// TIA Portal V17 export
// export: Created 2022-07-28T18:02:49.0040858Z, ExportSetting None, DisplayName Totally Integrated Automation Portal, DisplayVersion V17, DisplayName TIA Portal Openness, DisplayVersion V17, DisplayName TIA Portal Teamcenter Gateway, DisplayVersion V17, DisplayName TIA Portal Version Control Interface, DisplayVersion V17, DisplayName TIA Portal Test Suite Advanced, DisplayVersion V17, DisplayName SINAMICS Startdrive Advanced, DisplayVersion V17, DisplayName SINAMICS DCC, DisplayVersion V17, DisplayName SINAMICS Startdrive G130, G150, S120, S150, SINAMICS MV, S210, DisplayVersion V17, DisplayName SINAMICS Startdrive G110M, G120, G120C, G120D, G120P, G115D, DisplayVersion V17, DisplayName STEP 7 Professional, DisplayVersion V17, DisplayName SIMATIC Energy Suite, DisplayVersion V17, DisplayName STEP 7 CFC, DisplayVersion V17, DisplayName STEP 7 Safety, DisplayVersion V17, DisplayName WinCC Advanced / Unified PC, DisplayVersion V17, DisplayName SIMATIC Visualization Architect, DisplayVersion V17
FUNCTION_BLOCK "Lib_FB_PID_Cascad"   // FB151, SCL
{ S7_Optimized_Access := 'TRUE' }
// stored: AutoNumber false, MemoryReserve 100, SetENOAutomatically false
   VAR_INPUT
      I_Initialization { ExternalAccessible := 'False'; ExternalVisible := 'False'; ExternalWritable := 'False'} : Bool := FALSE;   // 1 = Restart PLC is active (First scan)
      IR_CycleTime { ExternalAccessible := 'False'; ExternalVisible := 'False'; ExternalWritable := 'False'} : Real := 0.0;   // Time of last PLC cycle, sec
      II_Obj_ID { ExternalAccessible := 'False'; ExternalVisible := 'False'; ExternalWritable := 'False'} : Int := -1;   // Tech ID of object
      I_CmdGeneralReset { ExternalAccessible := 'False'; ExternalVisible := 'False'; ExternalWritable := 'False'} : Bool;   // 0 ⮥ 1 = Input general reset ERROR/Interlocks
      I_One_1s { ExternalAccessible := 'False'; ExternalVisible := 'False'; ExternalWritable := 'False'} : Bool;   // 1 = One cycle per one seccond pulse
      I_EstopHMI { ExternalAccessible := 'False'; ExternalVisible := 'False'; ExternalWritable := 'False'} : Bool := TRUE;   // 0 = HMI/WinCC Emergency stop active
      IR_SP_Auto { ExternalAccessible := 'False'; ExternalVisible := 'False'; ExternalWritable := 'False'} : Real;   // SP for auto mode from input in physics units
      IR_MinOut { ExternalAccessible := 'False'; ExternalVisible := 'False'; ExternalWritable := 'False'} : Real := 15.0;   // Minimum output of PID, PU
      IR_MaxOut { ExternalAccessible := 'False'; ExternalVisible := 'False'; ExternalWritable := 'False'} : Real := 100.0;   // Maximum output of PID, PU
      IB_InterlocksOpen_8 { ExternalAccessible := 'False'; ExternalVisible := 'False'; ExternalWritable := 'False'} : Byte;   // <>0 = Interlock active - One or more from 8 Interlocks active // 1bit <--> 1 Interlock
      IB_InterlocksClose_8 { ExternalAccessible := 'False'; ExternalVisible := 'False'; ExternalWritable := 'False'} : Byte;   // <>0 = Interlock active - One or more from 8 Interlocks active // 1bit <--> 1 Interlock
      IW_ExternalError_16 { ExternalAccessible := 'False'; ExternalVisible := 'False'; ExternalWritable := 'False'} : Word;   // <>0 = External error active - One or more from 16 error active // 1bit <--> 1 error
      I_ExternalWarning { ExternalAccessible := 'False'; ExternalVisible := 'False'; ExternalWritable := 'False'} : Bool;   // 1 = External Warning
      IR_CyclePID { ExternalAccessible := 'False'; ExternalVisible := 'False'; ExternalWritable := 'False'} : Real;   // Cycle tyme of PID, sec
      II_ID_Sensor { ExternalAccessible := 'False'; ExternalVisible := 'False'; ExternalWritable := 'False'} : Int := -1;   // ID of sensor for PID
      IA_ID_Inv { ExternalAccessible := 'False'; ExternalVisible := 'False'; ExternalWritable := 'False'} : Array[0..5] of Int;   // IDs of inverters for PID
      II_Num_Inv { ExternalAccessible := 'False'; ExternalVisible := 'False'; ExternalWritable := 'False'} : Int := 3;   // Numbers of inverters
   END_VAR
   VAR_OUTPUT
      QR_Out_PID { ExternalAccessible := 'False'; ExternalVisible := 'False'; ExternalWritable := 'False'} : Real;   // Output of PID in physics unit (0-100%)
      QI_Out_PID { ExternalAccessible := 'False'; ExternalVisible := 'False'; ExternalWritable := 'False'} : Int;   // Output of PID in analog output units (0-27648)
      Q_CmdPWM { ExternalAccessible := 'False'; ExternalVisible := 'False'; ExternalWritable := 'False'} : Bool;   // PWM signal for descrete output mechanism
      Q_Reset { ExternalAccessible := 'False'; ExternalVisible := 'False'; ExternalWritable := 'False'} : Bool;   // 1 = Reset faults
      Q_Error { ExternalAccessible := 'False'; ExternalVisible := 'False'; ExternalWritable := 'False'} : Bool;   // This output indicates whether theres an error/fault condition in the motor
      Q_Auto { ExternalAccessible := 'False'; ExternalVisible := 'False'; ExternalWritable := 'False'} : Bool;   // 1= Automatic operating mode active
      Q_DataErr { ExternalAccessible := 'False'; ExternalVisible := 'False'; ExternalWritable := 'False'} : Bool;   // 1 = Transfer data error occured (ObjDB -> temp, ect)
   END_VAR
   VAR_IN_OUT
      IQ_PLC_CycleInfo : Variant;   // Ref to data about PLC cycle
   END_VAR
   VAR
      s_ErrForSwitchToOff { ExternalAccessible := 'False'; ExternalVisible := 'False'; ExternalWritable := 'False'} : Bool;   // 1 = Err occured for switch to manual mode
   END_VAR
   VAR RETAIN
      si_OldPriority_P1 { ExternalAccessible := 'False'; ExternalVisible := 'False'; ExternalWritable := 'False'} : Int := 1;
      si_OldPriority_P2 { ExternalAccessible := 'False'; ExternalVisible := 'False'; ExternalWritable := 'False'} : Int := 2;
      si_OldPriority_P3 { ExternalAccessible := 'False'; ExternalVisible := 'False'; ExternalWritable := 'False'} : Int := 3;
   END_VAR
   VAR
      si_CurrentPIDPoint { ExternalAccessible := 'False'; ExternalVisible := 'False'; ExternalWritable := 'False'} : Int;
      si_PrevPIDPoint { ExternalAccessible := 'False'; ExternalVisible := 'False'; ExternalWritable := 'False'} : Int;
      s_EdgeAuto { ExternalAccessible := 'False'; ExternalVisible := 'False'; ExternalWritable := 'False'} : "Lib_FB_Edge";
      s_EdgeMan { ExternalAccessible := 'False'; ExternalVisible := 'False'; ExternalWritable := 'False'} : "Lib_FB_Edge";
      s_EdgeOff { ExternalAccessible := 'False'; ExternalVisible := 'False'; ExternalWritable := 'False'} : "Lib_FB_Edge";
      s_EdgeSim { ExternalAccessible := 'False'; ExternalVisible := 'False'; ExternalWritable := 'False'} : "Lib_FB_Edge";
      s_EdgeError { ExternalAccessible := 'False'; ExternalVisible := 'False'; ExternalWritable := 'False'} : "Lib_FB_Edge";
      s_EdgeWarning { ExternalAccessible := 'False'; ExternalVisible := 'False'; ExternalWritable := 'False'} : "Lib_FB_Edge";
      s_EdgeUp { ExternalAccessible := 'False'; ExternalVisible := 'False'; ExternalWritable := 'False'} : "Lib_FB_Edge";
      s_EdgeDwn { ExternalAccessible := 'False'; ExternalVisible := 'False'; ExternalWritable := 'False'} : "Lib_FB_Edge";
   END_VAR
   VAR RETAIN
      s_Simulation { ExternalAccessible := 'False'; ExternalVisible := 'False'; ExternalWritable := 'False'} : Struct   // Data for simulation process
         Obj_DATA_BACKUP : Struct   // MOTOR NORMAL MODE DATA BACKUP FOR SIMULATION MODE
            Config : "_PID_Cascad_Config";
            Counters : "_PID_Cascad_Counters";
            sud_MotoHours_Electro : "_MotoHours_One";
            sud_MotoHours_Mech : "_MotoHours_One";
         END_STRUCT;
      END_STRUCT;
      s_Obj_Retain_BUp { ExternalAccessible := 'False'; ExternalVisible := 'False'; ExternalWritable := 'False'} : Struct
         Config : "_PID_Cascad_Config";
         Counters : "_PID_Cascad_Counters";
         Mode : "UDT_Mode";
      END_STRUCT;
   END_VAR
   VAR
      s_TP_ResetOut { ExternalAccessible := 'False'; ExternalVisible := 'False'; ExternalWritable := 'False'} : "Lib_FB_Timer_TP_Simple";
      s_TON_TimeUP { ExternalAccessible := 'False'; ExternalVisible := 'False'; ExternalWritable := 'False'} : "Lib_FB_Timer_ON_Simple";
      s_TON_TimeDwn { ExternalAccessible := 'False'; ExternalVisible := 'False'; ExternalWritable := 'False'} : "Lib_FB_Timer_ON_Simple";
      s_TON_Stabilization { ExternalAccessible := 'False'; ExternalVisible := 'False'; ExternalWritable := 'False'} : "Lib_FB_Timer_ON_Simple";
   END_VAR
   VAR_TEMP
      t_DataErr : Bool;   // 1 = Transfer data error occured (ObjDB -> temp, ect)
      t_ReleaseStart : Bool;   // 1 = Release for start in any mode
      t_SomePumpIsRunning : Bool;
      t_ResetLogic : Bool;   // 1 = Reset all signals for logic
      ti_CMDLogic : Int;   // Command word for logic
      ti_Cnt : Int;   // Counter for internal use
      ti_NumObjDB : UInt;   // Number of DB for storage object data
      t_MaxObjects : UInt;   // Max number of objects in plant
      tr_PID_Out : Real;   // SP in auto mode for logic
      tr_InvertCoef : Real;
      t_ObjAny_PIDCon : DB_ANY;
      t_ObjVar_PIDCon : Variant;
      t_ObjAny_HMI : DB_ANY;   // Ref to object data
      t_ObjVar_HMI : Variant;   // Ref to object data
      t_ObjAny_PLC : DB_ANY;   // Ref to object data
      t_ObjVar_PLC : Variant;   // Ref to object data
      t_SensorObjAny_HMI : DB_ANY;   // Ref to object data
      t_SensorObjVar_HMI : Variant;   // Ref to object data
      t_Pump1_ObjAny_HMI : DB_ANY;   // Ref to object data
      t_Pump1_ObjVar_HMI : Variant;   // Ref to object data
      t_Pump2_ObjAny_HMI : DB_ANY;   // Ref to object data
      t_Pump2_ObjVar_HMI : Variant;   // Ref to object data
      t_Pump3_ObjAny_HMI : DB_ANY;   // Ref to object data
      t_Pump3_ObjVar_HMI : Variant;   // Ref to object data
      t_PB_HMI : Struct   // Buttons from HMI
         ResetError : Bool;   // + set-->CMD_ALMACK_tag -Reset errors pushbutton
         AllInAuto : Bool;   // 1 = All pumps switch to auto
         spare2 : Bool;
         spare3 : Bool;
         spare4 : Bool;
         spare5 : Bool;
         spare6 : Bool;
         spare7 : Bool;
         spare8 : Bool;
         spare9 : Bool;
         spare10 : Bool;
         spare11 : Bool;
         spare12 : Bool;
         spare13 : Bool;
         spare14 : Bool;
         spare15 : Bool;
         spare16 : Bool;
         spare17 : Bool;
         spare18 : Bool;
         spare19 : Bool;
         spare20 : Bool;
         spare21 : Bool;
         spare22 : Bool;
         spare23 : Bool;
         spare24 : Bool;
         spare25 : Bool;
         spare26 : Bool;
         spare27 : Bool;
         spare28 : Bool;
         spare29 : Bool;
         spare30 : Bool;
         spare31 : Bool;
      END_STRUCT;
      t_Obj_HMI : "Lib_UDT_PID_Cascad_HMI";   // Object data
      t_Obj_PLC : "Lib_UDT_PID_Cascad_PLC";   // Object data
      t_Obj_PIDCon : "Lib_UDT_PID_Core";
      t_SensorObj_HMI : "lib_udt_ASensor_HMI";   // Object data
      t_Pump1_Obj_HMI : "Lib_UDT_Pump_Inv352_Base_HMI";   // Object data
      t_Pump2_Obj_HMI : "Lib_UDT_Pump_Inv352_Base_HMI";   // Object data
      t_Pump3_Obj_HMI : "Lib_UDT_Pump_Inv352_Base_HMI";   // Object data
      t_PLC_CycleInfo : "Lib_PLC_CycleInfo";   // Data about PLC cycle
      t_AutoControl : "Lib_UDT_AutoControl";   // Data for auto control module for current element
      t_AutoControl_Pumps : "_PID_Cascad_AutoCtrlPumpsAll";   // Data for auto control module for current element
      t_AutoControl_Pumps_Sorted : "_PID_Cascad_AutoCtrlPumpsAll";   // Data for auto control module for current element
      t_InternalData : "Lib_UDT_Int";   // Internal data
      t_Buffer : Array[0..100] of Byte;   // Buffer for use serialize
      tui_DB_ShiftHMI : UInt;   // Object DB number shift
      tui_DB_ShiftPLC : UInt;   // Object DB number shift
      tui_DB_ShiftPID : UInt;
   END_VAR
   // IA_ID_Inv[0..5] := -1;
BEGIN
   REGION Initialization/read data from out DB
       //Set internal data
       "Lib_FC_GenMoto_InitInternal"(#t_InternalData);

       //Reinit gen data
       #t_DataErr := false;
       #t_Obj_HMI.Config.w_enableExternalErrors_16 := w#16#FFFF;
       #t_Obj_HMI.Config.b_bypassInterlocksForward_8 := b#16#ff;
       #t_Obj_HMI.Config.b_bypassInterlocksReverse_8 := b#16#ff;
       #t_MaxObjects := "D_General_ProgramDATA".ui_MaxObjects;
       #tui_DB_ShiftHMI := "D_General_ProgramDATA".ui_Shift_DB_HMI;
       #tui_DB_ShiftPLC := "D_General_ProgramDATA".ui_Shift_DB_PLC;
       #tui_DB_ShiftPID := "D_General_ProgramDATA".ui_Shift_DB_PID;
       #t_AutoControl := "DB_AutoControl_arr".AutoControl_arr[#t_MaxObjects];
       #t_AutoControl_Pumps.Arr[0].AutoControl_P := "DB_AutoControl_arr".AutoControl_arr[#t_MaxObjects];
       #t_AutoControl_Pumps.Arr[1].AutoControl_P := "DB_AutoControl_arr".AutoControl_arr[#t_MaxObjects];
       #t_AutoControl_Pumps.Arr[2].AutoControl_P := "DB_AutoControl_arr".AutoControl_arr[#t_MaxObjects];

       //Read data PLC
       VariantGet(SRC := #IQ_PLC_CycleInfo,
                  DST => #t_PLC_CycleInfo);

       //Read Object data
       //Reinit temp values
       #t_Obj_HMI := "D_ZeroTypes".PID_Cascad_HMI;
       #t_Obj_PLC := "D_ZeroTypes".PID_Cascad_PLC;
       #t_SensorObj_HMI := "D_ZeroTypes".ASensor_HMI;
       #t_Pump1_Obj_HMI := "D_ZeroTypes".Pump_Inv352_Base_HMI;
       #t_Pump2_Obj_HMI := "D_ZeroTypes".Pump_Inv352_Base_HMI;
       #t_Pump3_Obj_HMI := "D_ZeroTypes".Pump_Inv352_Base_HMI;
       #t_Obj_PIDCon := "D_ZeroTypes".PID_Core;

       //Read object data
       IF #II_Obj_ID >= 0
       THEN
           //Read HMI data
           #ti_NumObjDB := INT_TO_UINT(#II_Obj_ID) + #tui_DB_ShiftHMI;
           #t_ObjAny_HMI := UINT_TO_DB_ANY(#ti_NumObjDB);
           #t_ObjVar_HMI := DB_ANY_TO_VARIANT(in := #t_ObjAny_HMI, err => #t_InternalData.i_Tmp);

           //If DB exist and convertion without error
           IF #t_InternalData.i_Tmp = 0
           THEN
               VariantGet(SRC := #t_ObjVar_HMI,
                          DST => #t_Obj_HMI);
           ELSE
               #t_DataErr := true;
           END_IF;

           //Read PLC data
           #ti_NumObjDB := INT_TO_UINT(#II_Obj_ID) + #tui_DB_ShiftPLC;
           #t_ObjAny_PLC := UINT_TO_DB_ANY(#ti_NumObjDB);
           #t_ObjVar_PLC := DB_ANY_TO_VARIANT(in := #t_ObjAny_PLC, err => #t_InternalData.i_Tmp);

           //If DB exist and convertion without error
           IF #t_InternalData.i_Tmp = 0
           THEN
               VariantGet(SRC := #t_ObjVar_PLC,
                          DST => #t_Obj_PLC);
           ELSE
               #t_DataErr := true;
           END_IF;

           //Read PID data
           #ti_NumObjDB := INT_TO_UINT(#II_Obj_ID) + #tui_DB_ShiftPID;
           #t_ObjAny_PIDCon := UINT_TO_DB_ANY(#ti_NumObjDB);
           #t_ObjVar_PIDCon := DB_ANY_TO_VARIANT(in := #t_ObjAny_PIDCon, err => #t_InternalData.i_Tmp);

           //If DB exist and convertion without error
           IF #t_InternalData.i_Tmp = 0
           THEN
               VariantGet(SRC := #t_ObjVar_PIDCon,
                          DST => #t_Obj_PIDCon);
           ELSE
               #t_DataErr := true;
           END_IF;
       ELSE
           #t_DataErr := true;
       END_IF;

       //Read sensor data
       IF #II_ID_Sensor >= 0
           AND NOT #t_DataErr
       THEN
           //Read HMI data
           #ti_NumObjDB := INT_TO_UINT(#II_ID_Sensor) + 50000;
           #t_SensorObjAny_HMI := UINT_TO_DB_ANY(#ti_NumObjDB);
           #t_SensorObjVar_HMI := DB_ANY_TO_VARIANT(in := #t_SensorObjAny_HMI, err => #t_InternalData.i_Tmp);

           //If DB exist and convertion without error
           IF #t_InternalData.i_Tmp = 0
           THEN
               VariantGet(SRC := #t_SensorObjVar_HMI,
                          DST => #t_SensorObj_HMI);
           ELSE
               #t_DataErr := true;
           END_IF;
       ELSE
           #t_DataErr := true;
       END_IF;

       //Read pumps data
       IF #IA_ID_Inv[0] >= 0
           AND NOT #t_DataErr
       THEN
           REGION Pump 1
               //Read HMI data
               #ti_NumObjDB := INT_TO_UINT(#IA_ID_Inv[0]) + #tui_DB_ShiftHMI;
               #t_Pump1_ObjAny_HMI := UINT_TO_DB_ANY(#ti_NumObjDB);
               #t_Pump1_ObjVar_HMI := DB_ANY_TO_VARIANT(in := #t_Pump1_ObjAny_HMI, err => #t_InternalData.i_Tmp);

               //If DB exist and convertion without error
               IF #t_InternalData.i_Tmp = 0
               THEN
                   VariantGet(SRC := #t_Pump1_ObjVar_HMI,
                              DST => #t_Pump1_Obj_HMI);
               ELSE
                   #t_DataErr := true;
               END_IF;

               #t_AutoControl_Pumps.Arr[0].AutoControl_P := "DB_AutoControl_arr".AutoControl_arr[#IA_ID_Inv[0]];
               #t_AutoControl_Pumps.Arr[0].i_IndexInArr := 0;
           END_REGION

       ELSE
           #t_DataErr := true;
       END_IF;

       IF #IA_ID_Inv[1] >= 0
           AND NOT #t_DataErr
       THEN
           REGION Pump 2
               //Read HMI data
               #ti_NumObjDB := INT_TO_UINT(#IA_ID_Inv[1]) + #tui_DB_ShiftHMI;
               #t_Pump2_ObjAny_HMI := UINT_TO_DB_ANY(#ti_NumObjDB);
               #t_Pump2_ObjVar_HMI := DB_ANY_TO_VARIANT(in := #t_Pump2_ObjAny_HMI, err => #t_InternalData.i_Tmp);

               //If DB exist and convertion without error
               IF #t_InternalData.i_Tmp = 0
               THEN
                   VariantGet(SRC := #t_Pump2_ObjVar_HMI,
      DST => #t_Pump2_Obj_HMI);
               ELSE
                   #t_DataErr := true;
               END_IF;

               #t_AutoControl_Pumps.Arr[1].AutoControl_P := "DB_AutoControl_arr".AutoControl_arr[#IA_ID_Inv[1]];
               #t_AutoControl_Pumps.Arr[1].i_IndexInArr := 1;
           END_REGION

       ELSE
           #t_DataErr := true;
       END_IF;

       IF #IA_ID_Inv[2] >= 0
           AND NOT #t_DataErr
       THEN
           REGION Pump 3
               //Read HMI data
               #ti_NumObjDB := INT_TO_UINT(#IA_ID_Inv[2]) + #tui_DB_ShiftHMI;
               #t_Pump3_ObjAny_HMI := UINT_TO_DB_ANY(#ti_NumObjDB);
               #t_Pump3_ObjVar_HMI := DB_ANY_TO_VARIANT(in := #t_Pump3_ObjAny_HMI, err => #t_InternalData.i_Tmp);

               //If DB exist and convertion without error
               IF #t_InternalData.i_Tmp = 0
               THEN
                   VariantGet(SRC := #t_Pump3_ObjVar_HMI,
      DST => #t_Pump3_Obj_HMI);
               ELSE
                   #t_DataErr := true;
               END_IF;

               #t_AutoControl_Pumps.Arr[2].AutoControl_P := "DB_AutoControl_arr".AutoControl_arr[#IA_ID_Inv[2]];
               #t_AutoControl_Pumps.Arr[2].i_IndexInArr := 2;
           END_REGION
       ELSE
           #t_DataErr := true;
       END_IF;

       //Read general info data
       CASE #II_Obj_ID OF
           0..999:  // ID of element in range
               #t_AutoControl := "DB_AutoControl_arr".AutoControl_arr[#II_Obj_ID];
           ELSE
               ;
       END_CASE;

       //Read retain data if initialization is active
       IF #I_Initialization
       THEN
           #t_Obj_HMI.Config := #s_Obj_Retain_BUp.Config;
           #t_Obj_HMI.Counters := #s_Obj_Retain_BUp.Counters;
           #t_Obj_PLC.Mode := #s_Obj_Retain_BUp.Mode;
       END_IF;
   END_REGION
   //---------------------------------------------------------------
   //---------------------------------------------------------------
   REGION Check ranges
       //Invert coef
       IF #t_Obj_HMI.Config.b.DirectMode
       THEN
           #tr_InvertCoef := 1.0;
       ELSE
           #tr_InvertCoef := -1.0;
       END_IF;

       IF #t_Obj_HMI.Config.r_FTC_Value > #IR_MaxOut
       THEN
           #t_Obj_HMI.Config.r_FTC_Value := #IR_MaxOut;
       END_IF;

       IF #t_Obj_HMI.Config.r_FTC_Value < #IR_MinOut
       THEN
           #t_Obj_HMI.Config.r_FTC_Value := #IR_MinOut;
       END_IF;

       IF #t_Obj_HMI.Config.r_SP_Auto_Value > #t_SensorObj_HMI.Config.r_MaxVal
       THEN
           #t_Obj_HMI.Config.r_SP_Auto_Value := #t_SensorObj_HMI.Config.r_MaxVal;
       END_IF;

       IF #t_Obj_HMI.Config.r_SP_Auto_Value < #t_SensorObj_HMI.Config.r_MinVal
       THEN
           #t_Obj_HMI.Config.r_SP_Auto_Value := #t_SensorObj_HMI.Config.r_MinVal;
       END_IF;
   END_REGION
   //---------------------------------------------------------------
   //---------------------------------------------------------------
   REGION Define CMD for block logic 
       //Reinit logic CMD
       #ti_CMDLogic := 0;

       "Lib_FC_GenMoto_ChoiceCMD"(I_Mode := #t_Obj_PLC.Mode,
                                  QI_CMD_Logic => #ti_CMDLogic,
                                  IQI_CMD_Global := #t_PLC_CycleInfo.CMD_GLOBAL,
                                  IQI_CMD_Auto := #t_AutoControl.Global_CMD,
                                  IQI_CMD_HMI := #t_Obj_HMI.i_CMD);

   END_REGION
   //---------------------------------------------------------------
   //---------------------------------------------------------------
   REGION Switch modes  
       "Lib_FC_GenMoto_SwitchMode"(I_ManLocalModeActive := false,
                                   IQI_CMD_Logic := #ti_CMDLogic,
                                   IQ_Mode := #t_Obj_PLC.Mode,
                                   IQ_ObjDataConfig := #t_Obj_HMI.Config,
                                   IQ_BUpDataConfig := #s_Simulation.Obj_DATA_BACKUP.Config,
                                   IQ_ObjDataCounters := #t_Obj_HMI.Counters,
                                   IQ_BUpDataCounters := #s_Simulation.Obj_DATA_BACKUP.Counters);
                                END_REGION
   //---------------------------------------------------------------
   //---------------------------------------------------------------
   REGION Forcely switch modes by mode of PID  
      (* 
       IF (NOT (#t_Obj_PIDCon.i_State = 4)
           AND NOT (#t_Obj_PIDCon.i_State = 3))
           OR #s_ErrForSwitchToOff
       THEN
           #ti_CMDLogic := 1;
       END_IF;

       "Lib_FC_GenMoto_SwitchMode"(I_ManLocalModeActive := false,
                                   IQI_CMD_Logic := #ti_CMDLogic,
                                   IQ_Mode := #t_Obj_PLC.Mode,
                                   IQ_ObjDataConfig := #t_Obj_HMI.Config,
                                   IQ_BUpDataConfig := #s_Simulation.Obj_DATA_BACKUP.Config,
                                   IQ_ObjDataCounters := #t_Obj_HMI.Counters,
                                   IQ_BUpDataCounters := #s_Simulation.Obj_DATA_BACKUP.Counters); *)
   END_REGION
   //---------------------------------------------------------------
   //---------------------------------------------------------------
   REGION Convert commands to bit
       //Reinit all bits
       SCATTER(IN := #t_InternalData.d_Alw0,
               OUT => #t_PB_HMI);

       //Read commands and set apropriate bits
       CASE #ti_CMDLogic OF
           22:  //Direct mode
               #t_Obj_HMI.Config.b.DirectMode := true;
           23:  //Invert mode
               #t_Obj_HMI.Config.b.DirectMode := false;
           24:  //Invert mode
               #t_Obj_HMI.Config.b.Enabled_P1 := true;
           25:  //Invert mode
               #t_Obj_HMI.Config.b.Enabled_P2 := true;
           26:  //Invert mode
               #t_Obj_HMI.Config.b.Enabled_P3 := true;
           27:  //Invert mode
               #t_Obj_HMI.Config.b.Enabled_P1 := false;
           28:  //Invert mode
               #t_Obj_HMI.Config.b.Enabled_P2 := false;
           29:  //Invert mode
               #t_Obj_HMI.Config.b.Enabled_P3 := false;
           31..32: // Reset errors
               #t_PB_HMI.ResetError := true;
           30:// Switch all pumps to auto
               #t_PB_HMI.AllInAuto := true;

           ELSE
               ;
       END_CASE;

       //General bits for logic
       //General reset
       #t_ResetLogic := #t_PB_HMI.ResetError
       OR #I_CmdGeneralReset;

       //Reset for out of block
       #s_TP_ResetOut(IR_CycleTime := #IR_CycleTime,
                      IB_StartTimerInput := #t_ResetLogic,
                      IR_SpTime := 1.5);

                   END_REGION
   //---------------------------------------------------------------
   //---------------------------------------------------------------
   REGION Switch mode on PID
       //Catch change mode
       #s_EdgeAuto(IB_Input := #t_Obj_PLC.Mode.Auto);
       #s_EdgeMan(IB_Input := #t_Obj_PLC.Mode.ManualRemote);
       #s_EdgeOff(IB_Input := #s_ErrForSwitchToOff);

       IF #s_EdgeAuto.QB_EdgePos
           OR #s_EdgeMan.QB_EdgePos
           OR #s_EdgeOff.QB_EdgePos
       THEN
           #t_Obj_PIDCon.ModeActivate := true;
       END_IF;
       //Set value for auto mode
       IF (#s_EdgeAuto.QB_EdgePos
           AND #t_Obj_PIDCon.ModeActivate
           AND NOT (#t_Obj_PIDCon.i_State = 3))
       THEN
           #t_Obj_PIDCon.i_Mode := 3;
       END_IF;

       //Set value for manual mode
       IF (#s_EdgeMan.QB_EdgePos
           AND #t_Obj_PIDCon.ModeActivate
           AND NOT (#t_Obj_PIDCon.i_State = 4))
       THEN
           #t_Obj_PIDCon.i_Mode := 4;
       END_IF;

       //Set value for off mode
       IF (#s_EdgeOff.QB_EdgePos
           AND #t_Obj_PIDCon.ModeActivate
           AND NOT (#t_Obj_PIDCon.i_State = 0))
       THEN
           #t_Obj_PIDCon.i_Mode := 0;
       END_IF;
   END_REGION
   //---------------------------------------------------------------
   //---------------------------------------------------------------
   REGION Write data to PID and call him
       #t_Obj_PIDCon.r_Setpoint := #t_Obj_HMI.Config.r_SP_Auto_Value;
       #t_Obj_PIDCon.r_ManualValue := #t_Obj_HMI.Config.r_SP_Man_Value;
       #t_Obj_PIDCon.r_Input := #t_SensorObj_HMI.Config.r_DisplayData;
       IF #t_ResetLogic
       THEN
           #t_Obj_PIDCon.ErrorAck := true;
       END_IF;
       IF #I_Initialization
       THEN
           #t_Obj_PIDCon.Reset := true;
       END_IF;
       #t_Obj_PIDCon.r_OutputUpperLimit := #IR_MaxOut;
       #t_Obj_PIDCon.r_OutputLowerLimit := #IR_MinOut;
       #t_Obj_PIDCon.r_CycleTime_Value := #IR_CyclePID;
       #t_Obj_PIDCon.r_Gain := #tr_InvertCoef * #t_Obj_HMI.Config.r_spP_part;
       #t_Obj_PIDCon.r_Ti := #t_Obj_HMI.Config.r_spI_part;
       #t_Obj_PIDCon.r_Td := #t_Obj_HMI.Config.r_spD_part;
       #t_Obj_PIDCon.InvertControl := false; //NOT #t_Obj_HMI.Config.b.DirectMode;
       #t_Obj_PIDCon.r_SPUpperLimit := #t_SensorObj_HMI.Config.r_MaxVal;
       #t_Obj_PIDCon.r_SPLowerLimit := #t_SensorObj_HMI.Config.r_MinVal;
       #t_Obj_PIDCon.r_PVUpperLimit := #t_SensorObj_HMI.Config.r_MaxVal;
       #t_Obj_PIDCon.r_PVLowerLimit := #t_SensorObj_HMI.Config.r_MinVal;
       #t_Obj_PIDCon.r_Cycle_PID := 1.0;

       //Write mode by mode on PID
       #t_Obj_PLC.Mode.Auto := #t_Obj_PIDCon.i_State = 3;
       #t_Obj_PLC.Mode.ManualRemote := #t_Obj_PIDCon.i_State = 4;
       #t_Obj_PLC.Mode.Disable := #t_Obj_PIDCon.i_State = 0;

       REGION Store out of PID in temp var dependent of state
           IF #t_Obj_PIDCon.i_State = 3
               OR #t_Obj_PIDCon.i_State = 4
           THEN
               #tr_PID_Out := #t_Obj_PIDCon.r_Output;
           ELSE
               IF #t_Obj_PLC.State.FTCActive
               THEN
                   #tr_PID_Out := #t_Obj_HMI.Config.r_FTC_Value;
               ELSIF #t_Obj_PLC.State.FTOActive
               THEN
                   #tr_PID_Out := #t_Obj_HMI.Config.r_FTO_Value;
               ELSE
                   #tr_PID_Out := #IR_MinOut;
               END_IF;
           END_IF;
       END_REGION

   END_REGION
   //---------------------------------------------------------------
   //---------------------------------------------------------------
   REGION Control of pumps

       REGION Define number OF enabled pumps
           #t_Obj_HMI.Config.r_QuanEnabled := 0;

           IF #t_Obj_HMI.Config.b.Enabled_P1
           THEN
               #t_Obj_HMI.Config.r_QuanEnabled := #t_Obj_HMI.Config.r_QuanEnabled + 1;
           END_IF;
           IF #t_Obj_HMI.Config.b.Enabled_P2
           THEN
               #t_Obj_HMI.Config.r_QuanEnabled := #t_Obj_HMI.Config.r_QuanEnabled + 1;
           END_IF;
           IF #t_Obj_HMI.Config.b.Enabled_P3
           THEN
               #t_Obj_HMI.Config.r_QuanEnabled := #t_Obj_HMI.Config.r_QuanEnabled + 1;
           END_IF;

       END_REGION

       REGION Define priority of pumps
           IF #t_Obj_HMI.Config.b.Enabled_P1
           THEN
               IF #t_Obj_HMI.Config.i_Priority_P1 > #t_Obj_HMI.Config.r_QuanEnabled
               THEN
                   #t_Obj_HMI.Config.i_Priority_P1 := #t_Obj_HMI.Config.r_QuanEnabled;
                   #si_OldPriority_P1 := #t_Obj_HMI.Config.r_QuanEnabled;
               END_IF;
           ELSE
               #t_Obj_HMI.Config.i_Priority_P1 := #t_Obj_HMI.Config.r_QuanEnabled + 1;
               #si_OldPriority_P1 := #t_Obj_HMI.Config.r_QuanEnabled + 1;
           END_IF;
           IF #t_Obj_HMI.Config.b.Enabled_P2
           THEN
               IF #t_Obj_HMI.Config.i_Priority_P2 > #t_Obj_HMI.Config.r_QuanEnabled
               THEN
                   #t_Obj_HMI.Config.i_Priority_P2 := #t_Obj_HMI.Config.r_QuanEnabled;
                   #si_OldPriority_P2 := #t_Obj_HMI.Config.r_QuanEnabled;
               END_IF;
           ELSE
               #t_Obj_HMI.Config.i_Priority_P2 := #t_Obj_HMI.Config.r_QuanEnabled + 1;
               #si_OldPriority_P2 := #t_Obj_HMI.Config.r_QuanEnabled + 1;
           END_IF;
           IF #t_Obj_HMI.Config.b.Enabled_P3
           THEN
               IF #t_Obj_HMI.Config.i_Priority_P3 > #t_Obj_HMI.Config.r_QuanEnabled
               THEN
                   #t_Obj_HMI.Config.i_Priority_P3 := #t_Obj_HMI.Config.r_QuanEnabled;
                   #si_OldPriority_P3 := #t_Obj_HMI.Config.r_QuanEnabled;
               END_IF;
           ELSE
               #t_Obj_HMI.Config.i_Priority_P3 := #t_Obj_HMI.Config.r_QuanEnabled + 1;
               #si_OldPriority_P3 := #t_Obj_HMI.Config.r_QuanEnabled + 1;
           END_IF;

           //If priority the same
           IF #t_Obj_HMI.Config.i_Priority_P1 = #t_Obj_HMI.Config.i_Priority_P2
               AND #t_Obj_HMI.Config.i_Priority_P1 = #t_Obj_HMI.Config.i_Priority_P3
               AND #t_Obj_HMI.Config.b.Enabled_P1
               AND #t_Obj_HMI.Config.b.Enabled_P2
               AND #t_Obj_HMI.Config.b.Enabled_P3
           THEN
               #t_Obj_HMI.Config.i_Priority_P1 := 1;
               #t_Obj_HMI.Config.i_Priority_P2 := 2;
               #t_Obj_HMI.Config.i_Priority_P3 := 3;
               #si_OldPriority_P1 := 1;
               #si_OldPriority_P2 := 2;
               #si_OldPriority_P3 := 3;
           END_IF;

           //If priority changed
           REGION Changed priority for pump1
               IF NOT (#t_Obj_HMI.Config.i_Priority_P1 = 0)
               THEN
                   IF #t_Obj_HMI.Config.i_Priority_P1 <> #si_OldPriority_P1
                   THEN
                       IF #t_Obj_HMI.Config.i_Priority_P1 = #t_Obj_HMI.Config.i_Priority_P2
                           AND #t_Obj_HMI.Config.b.Enabled_P2
                       THEN
                           #t_Obj_HMI.Config.i_Priority_P2 := #si_OldPriority_P1;
                           #si_OldPriority_P2 := #si_OldPriority_P1;
                       END_IF;

                       IF #t_Obj_HMI.Config.i_Priority_P1 = #t_Obj_HMI.Config.i_Priority_P3
                           AND #t_Obj_HMI.Config.b.Enabled_P3
                       THEN
                           #t_Obj_HMI.Config.i_Priority_P3 := #si_OldPriority_P1;
                           #si_OldPriority_P3 := #si_OldPriority_P1;
                       END_IF;
                   END_IF;
               ELSE
                   #t_Obj_HMI.Config.i_Priority_P1 := 1;
               END_IF;
           END_REGION

           REGION Changed priority for pump2
               IF NOT (#t_Obj_HMI.Config.i_Priority_P2 = 0)
               THEN
                   IF #t_Obj_HMI.Config.i_Priority_P2 <> #si_OldPriority_P2
                   THEN
                       IF #t_Obj_HMI.Config.i_Priority_P2 = #t_Obj_HMI.Config.i_Priority_P1
                           AND #t_Obj_HMI.Config.b.Enabled_P1
                       THEN
                           #t_Obj_HMI.Config.i_Priority_P1 := #si_OldPriority_P2;
                           #si_OldPriority_P1 := #si_OldPriority_P2;
                       END_IF;

                       IF #t_Obj_HMI.Config.i_Priority_P2 = #t_Obj_HMI.Config.i_Priority_P3
                           AND #t_Obj_HMI.Config.b.Enabled_P3
                       THEN
                           #t_Obj_HMI.Config.i_Priority_P3 := #si_OldPriority_P2;
                           #si_OldPriority_P3 := #si_OldPriority_P2;
                       END_IF;
                   END_IF;
               ELSE
                   #t_Obj_HMI.Config.i_Priority_P2 := 2;
               END_IF;
           END_REGION

           REGION Changed priority for pump3
               IF NOT (#t_Obj_HMI.Config.i_Priority_P3 = 0)
               THEN
                   IF #t_Obj_HMI.Config.i_Priority_P3 <> #si_OldPriority_P3
                   THEN
                       IF #t_Obj_HMI.Config.i_Priority_P3 = #t_Obj_HMI.Config.i_Priority_P2
                           AND #t_Obj_HMI.Config.b.Enabled_P2
                       THEN
                           #t_Obj_HMI.Config.i_Priority_P2 := #si_OldPriority_P3;
                           #si_OldPriority_P2 := #si_OldPriority_P3;
                       END_IF;

                       IF #t_Obj_HMI.Config.i_Priority_P3 = #t_Obj_HMI.Config.i_Priority_P1
                           AND #t_Obj_HMI.Config.b.Enabled_P3
                       THEN
                           #t_Obj_HMI.Config.i_Priority_P1 := #si_OldPriority_P3;
                           #si_OldPriority_P1 := #si_OldPriority_P3;
                       END_IF;
                   END_IF;
               ELSE
                   #t_Obj_HMI.Config.i_Priority_P3 := 3;
               END_IF;
           END_REGION

           #si_OldPriority_P1 := #t_Obj_HMI.Config.i_Priority_P1;
           #si_OldPriority_P2 := #t_Obj_HMI.Config.i_Priority_P2;
           #si_OldPriority_P3 := #t_Obj_HMI.Config.i_Priority_P3;

           #t_AutoControl_Pumps.Arr[0].i_Priority := #t_Obj_HMI.Config.i_Priority_P1;
           #t_AutoControl_Pumps.Arr[1].i_Priority := #t_Obj_HMI.Config.i_Priority_P2;
           #t_AutoControl_Pumps.Arr[2].i_Priority := #t_Obj_HMI.Config.i_Priority_P3;

           #t_AutoControl_Pumps.Arr[0].Enabled := #t_Obj_HMI.Config.b.Enabled_P1;
           #t_AutoControl_Pumps.Arr[1].Enabled := #t_Obj_HMI.Config.b.Enabled_P2;
           #t_AutoControl_Pumps.Arr[2].Enabled := #t_Obj_HMI.Config.b.Enabled_P3;
       END_REGION

       #t_AutoControl_Pumps_Sorted := "Lib_FC_PID_Cascad_SortPrior"(#t_AutoControl_Pumps);
       #t_InternalData.i_Tmp := #t_AutoControl_Pumps_Sorted.Arr[0].i_IndexInArr;
       #t_InternalData.i_Tmp := #t_AutoControl_Pumps_Sorted.Arr[1].i_IndexInArr;
       #t_InternalData.i_Tmp := #t_AutoControl_Pumps_Sorted.Arr[2].i_IndexInArr;

       REGION Define current, next and prev points
           //Some of pumps is running
           #t_SomePumpIsRunning := #t_AutoControl_Pumps.Arr[0].AutoControl_P.StatusGen.ControlAchieve
           OR #t_AutoControl_Pumps.Arr[1].AutoControl_P.StatusGen.ControlAchieve
           OR #t_AutoControl_Pumps.Arr[2].AutoControl_P.StatusGen.ControlAchieve;

           IF NOT #t_SomePumpIsRunning
           THEN
               "Lib_FC_PID_Cascad_SetInitPID"(#t_AutoControl_Pumps_Sorted);
           ELSE
               //Define points for go up
               IF #s_EdgeUp.QB_EdgePos
               THEN
                   #si_CurrentPIDPoint := "Lib_FC_PID_Cascad_AddNextPID"(#t_AutoControl_Pumps_Sorted);

                   IF #si_CurrentPIDPoint <> #si_PrevPIDPoint
                   THEN

                       #t_InternalData.r_Tmp := #t_Obj_PIDCon.r_Gain * (#t_Obj_PIDCon.r_Setpoint - #t_Obj_PIDCon.r_Input);
                       #t_InternalData.r_Tmp := #IR_MinOut - #t_InternalData.r_Tmp;

                       IF #t_Obj_PIDCon.r_Gain <> 0.0
                       THEN
                           #t_Obj_PIDCon.r_IntegralSum := #t_InternalData.r_Tmp / #t_Obj_PIDCon.r_Gain;
                       ELSE
                           #t_Obj_PIDCon.r_IntegralSum  := #IR_MinOut;
                       END_IF;

                      // #t_Obj_PIDCon.r_IntegralSum := #IR_MinOut - #t_Obj_PIDCon.r_Gain * (#t_Obj_PIDCon.r_Setpoint - #t_Obj_PIDCon.r_Input);
                       #t_Obj_PIDCon.r_Output := #IR_MinOut;
                      #tr_PID_Out := #IR_MinOut;
                       #t_Obj_PIDCon.SetIntegralSum := true;
                       #si_PrevPIDPoint := #si_CurrentPIDPoint;
                   END_IF;
               END_IF;

               //Define points for go dwn
               IF #s_EdgeDwn.QB_EdgePos
               THEN
                   #si_CurrentPIDPoint := "Lib_FC_PID_Cascad_RemovePrevPID"(#t_AutoControl_Pumps_Sorted);

                   IF #si_CurrentPIDPoint <> #si_PrevPIDPoint
                   THEN
                       #t_InternalData.r_Tmp := #t_Obj_PIDCon.r_Gain * (#t_Obj_PIDCon.r_Setpoint - #t_Obj_PIDCon.r_Input);
                       #t_InternalData.r_Tmp := #IR_MaxOut - #t_InternalData.r_Tmp;

                       IF #t_Obj_PIDCon.r_Gain <> 0.0
                       THEN
                           #t_Obj_PIDCon.r_IntegralSum := #t_InternalData.r_Tmp / #t_Obj_PIDCon.r_Gain;
                       ELSE
                           #t_Obj_PIDCon.r_IntegralSum  := #IR_MaxOut;
                       END_IF;

                      // #t_Obj_PIDCon.r_IntegralSum := #IR_MaxOut - #t_Obj_PIDCon.r_Gain * (#t_Obj_PIDCon.r_Setpoint - #t_Obj_PIDCon.r_Input);
                       #tr_PID_Out := #IR_MaxOut;
                       #t_Obj_PIDCon.r_Output := #IR_MaxOut;
                       #t_Obj_PIDCon.SetIntegralSum := true;
                       #si_PrevPIDPoint := #si_CurrentPIDPoint;
                   END_IF;
               END_IF;

               //Recalc next PID if current not ready
               FOR #ti_Cnt := 0 TO 2 DO
                   IF #t_AutoControl_Pumps_Sorted.Arr[#ti_Cnt].AutoControl_P.StatusGen.StartPID
                       AND (NOT #t_AutoControl_Pumps_Sorted.Arr[#ti_Cnt].Enabled
                       OR NOT #t_AutoControl_Pumps_Sorted.Arr[#ti_Cnt].AutoControl_P.Mode.Auto
                       OR NOT #t_AutoControl_Pumps_Sorted.Arr[#ti_Cnt].AutoControl_P.StatusGen.Ready)
                   THEN
                       "Lib_FC_PID_Cascad_SetNextFreePID"(#t_AutoControl_Pumps_Sorted);
                   END_IF;
               END_FOR;

               //Recalc next Full if current not ready
               FOR #ti_Cnt := 0 TO 2 DO
                   IF #t_AutoControl_Pumps_Sorted.Arr[#ti_Cnt].AutoControl_P.StatusGen.StartFull
                       AND (NOT #t_AutoControl_Pumps_Sorted.Arr[#ti_Cnt].Enabled
                       OR NOT #t_AutoControl_Pumps_Sorted.Arr[#ti_Cnt].AutoControl_P.Mode.Auto
                       OR NOT #t_AutoControl_Pumps_Sorted.Arr[#ti_Cnt].AutoControl_P.StatusGen.Ready)
                   THEN
                       "Lib_FC_PID_Cascad_SetNextFreePID"(#t_AutoControl_Pumps_Sorted);
                   END_IF;
               END_FOR;
           END_IF;
       END_REGION

       REGION Timers and edges for go to next and previous points
           #s_TON_TimeUP(IR_CycleTime := #IR_CycleTime,
                         IB_StartTimerInput := #tr_PID_Out >= #IR_MaxOut
                         AND NOT #s_ErrForSwitchToOff
                         AND #t_SomePumpIsRunning,
                         IB_ResetTimer := #I_Initialization
                         OR #s_EdgeUp.QB_EdgePos,
                         IR_SpTime:=#t_Obj_HMI.Config.r_spCascadeTime);
           #s_TON_TimeDwn(IR_CycleTime := #IR_CycleTime,
                          IB_StartTimerInput := #tr_PID_Out <= #IR_MinOut
                          AND NOT #s_ErrForSwitchToOff
                          AND #t_SomePumpIsRunning,
                          IB_ResetTimer := #I_Initialization
                          OR #s_EdgeDwn.QB_EdgePos,
                          IR_SpTime:=#t_Obj_HMI.Config.r_spCascadeTime);
           #s_EdgeUp(IB_Input:=#s_TON_TimeUP.QB_TimerOut);
           #s_EdgeDwn(IB_Input:=#s_TON_TimeDwn.QB_TimerOut);
       END_REGION

       #t_AutoControl_Pumps := "Lib_FC_PID_Cascad_DeSortPrior"(#t_AutoControl_Pumps_Sorted);
       #t_InternalData.i_Tmp := #t_AutoControl_Pumps.Arr[0].i_IndexInArr;
       #t_InternalData.i_Tmp := #t_AutoControl_Pumps.Arr[1].i_IndexInArr;
       #t_InternalData.i_Tmp := #t_AutoControl_Pumps.Arr[2].i_IndexInArr;

       REGION Control of pumps
           FOR #ti_Cnt := 0 TO 2 DO
               IF NOT #t_AutoControl_Pumps.Arr[#ti_Cnt].Enabled
                   OR NOT #t_Obj_PLC.Mode.Auto
                   OR NOT #t_AutoControl_Pumps.Arr[#ti_Cnt].AutoControl_P.Mode.Auto
                   OR NOT #t_AutoControl_Pumps.Arr[#ti_Cnt].AutoControl_P.StatusGen.Ready
               THEN
                   #t_AutoControl_Pumps.Arr[#ti_Cnt].AutoControl_P.CTW.%X0 := false;
                   #t_AutoControl_Pumps.Arr[#ti_Cnt].AutoControl_P.SP_AutoMode := 0.0;
                   "Lib_FC_PID_Cascad_RemoveStart"(#t_AutoControl_Pumps.Arr[#ti_Cnt]);
               ELSE
                   #t_AutoControl_Pumps.Arr[#ti_Cnt].AutoControl_P.SP_AutoMode := 0.0;
                   #t_AutoControl_Pumps.Arr[#ti_Cnt].AutoControl_P.CTW.%X0 := #t_AutoControl_Pumps.Arr[#ti_Cnt].AutoControl_P.StatusGen.StartFull
                   OR #t_AutoControl_Pumps.Arr[#ti_Cnt].AutoControl_P.StatusGen.StartPID;

                   IF #t_AutoControl_Pumps.Arr[#ti_Cnt].AutoControl_P.StatusGen.StartFull
                   THEN
                       #t_AutoControl_Pumps.Arr[#ti_Cnt].AutoControl_P.SP_AutoMode := 100.0;
                   END_IF;

                   IF #t_AutoControl_Pumps.Arr[#ti_Cnt].AutoControl_P.StatusGen.StartPID
                   THEN
                       #t_AutoControl_Pumps.Arr[#ti_Cnt].AutoControl_P.SP_AutoMode := #tr_PID_Out;
                   END_IF;

               END_IF;
           END_FOR;
       END_REGION

       REGION Switch all pumps in auto
           FOR #ti_Cnt := 0 TO 2 DO
               IF #t_PB_HMI.AllInAuto
                   AND #t_AutoControl_Pumps.Arr[#ti_Cnt].Enabled
                   AND NOT #t_AutoControl_Pumps.Arr[#ti_Cnt].AutoControl_P.STW_HMI.%X25
               THEN
                   #t_AutoControl_Pumps.Arr[#ti_Cnt].AutoControl_P.Global_CMD := 2;
               END_IF;
           END_FOR;
       END_REGION

   END_REGION
   //---------------------------------------------------------------
   //---------------------------------------------------------------
   REGION Proccess faults, warnings, interlocks and status bits

       REGION Reinit words
           // Reinit alarm words
           IF #t_ResetLogic
               OR #I_Initialization
               OR #t_Obj_PLC.Mode.Disable
               OR #t_Obj_PLC.Mode.Repair
           THEN
               #t_Obj_HMI.Status.w_ALW1 := #t_InternalData.w_Alw0;
               #t_Obj_HMI.Status.w_ALW2 := #t_InternalData.w_Alw0;
               #t_Obj_HMI.Status.w_ALW3 := #t_InternalData.w_Alw0;
               #t_Obj_HMI.Status.w_ALW4 := #t_InternalData.w_Alw0;
               #t_Obj_HMI.Status.w_ALW5 := #t_InternalData.w_Alw0;
               //#t_Obj_PLC.State := "DB_ZeroTypes".PID_Cascad_PLC.State;
               #t_Obj_PLC.Alarm := "D_ZeroTypes".PID_Cascad_PLC.Alarm;
           END_IF;

           //Reinit STW words
           #t_Obj_HMI.Status.dw_STW := #t_InternalData.d_Alw0;

           //Reinit interlocks words
           #t_Obj_HMI.Status.dw_ILW_Frw := #t_InternalData.d_Alw0;
           #t_Obj_HMI.Status.dw_ILW_Rev := #t_InternalData.d_Alw0;
       END_REGION

       //Interlocks
       #t_Obj_PLC.State.FTCActive := ((#t_Obj_HMI.Config.b_bypassInterlocksForward_8
       AND #IB_InterlocksOpen_8) <> b#16#0)
       AND NOT #t_Obj_PLC.Mode.Disable
       AND NOT #t_Obj_PLC.Mode.Service;

       #t_Obj_PLC.State.FTOActive := ((#t_Obj_HMI.Config.b_bypassInterlocksReverse_8
       AND #IB_InterlocksClose_8) <> b#16#0)
       AND NOT #t_Obj_PLC.Mode.Disable
       AND NOT #t_Obj_PLC.Mode.Service;

       #t_Obj_HMI.Status.dw_ILW_Frw.%B0 := #IB_InterlocksOpen_8;
       #t_Obj_HMI.Status.dw_ILW_Rev.%B0 := #IB_InterlocksClose_8;

       REGION Faults common for sim and gen modes
           IF NOT #t_Obj_PLC.Mode.Disable
           THEN
               //Emergency stop from HMI 
               #t_Obj_PLC.Alarm.EstopHMI := NOT #I_EstopHMI;

               //External error
               #t_Obj_HMI.Status.dw_EEW.%W0 := #IW_ExternalError_16;
               #t_Obj_PLC.Alarm.ExtError := (#IW_ExternalError_16
               AND #t_Obj_HMI.Config.w_enableExternalErrors_16) <> w#16#0;

               //Sensor Err
               #t_Obj_PLC.Alarm.SensorErr := #t_SensorObj_HMI.Status.dw_STW.%X15;

               //Inverters err
               #t_Obj_PLC.Alarm.InverterErr := (#t_Pump1_Obj_HMI.Status.dw_STW.%X0
               AND #t_Obj_HMI.Status.dw_STW_P1.%X2)
               OR (#t_Pump2_Obj_HMI.Status.dw_STW.%X0
               AND #t_Obj_HMI.Status.dw_STW_P2.%X2)
               OR (#t_Pump3_Obj_HMI.Status.dw_STW.%X0
               AND #t_Obj_HMI.Status.dw_STW_P3.%X2);

               //PID err
               #t_Obj_PLC.Alarm.PIDErr := #t_Obj_PIDCon.Error;

               //FTC active
               #t_Obj_PLC.Alarm.FTCActive := #t_Obj_PLC.State.FTCActive;

               //FTO active
               #t_Obj_PLC.Alarm.FTOActive := #t_Obj_PLC.State.FTOActive;

               //HL active
               #t_Obj_PLC.Alarm.HLActive := #t_Obj_PIDCon.r_Output >= #IR_MaxOut;

               //LL active
               #t_Obj_PLC.Alarm.LLActive := #t_Obj_PIDCon.r_Output <= #IR_MinOut;

               //Stabilization err
               #t_Obj_PLC.Alarm.StabilizationErr := #s_TON_Stabilization.QB_TimerOut;

           END_IF;
       END_REGION

       REGION Faults different for gen and sim modes
           IF NOT #t_Obj_PLC.Mode.Simulation
               AND NOT #t_Obj_PLC.Mode.Disable
           THEN

               #t_Obj_PLC.Alarm := #t_Obj_PLC.Alarm;
           ELSIF #t_Obj_PLC.Mode.Simulation
               AND NOT #t_Obj_PLC.Mode.Disable
           THEN
               //CMD for test in simulation mode
               //Need remove line below
               #t_Obj_PLC.Alarm := #t_Obj_PLC.Alarm;

           END_IF;

           REGION Timers, edges ect.
               #s_TON_Stabilization(IR_CycleTime := #IR_CycleTime,
                                    IB_StartTimerInput := #t_Obj_PLC.Mode.Auto
                                    AND (ABS(#t_Obj_PIDCon.r_Input - #t_Obj_PIDCon.r_Setpoint) > 0.5),
                                    IB_ResetTimer := #I_Initialization
                                    OR #t_ResetLogic,
                                    IR_SpTime := #t_Obj_HMI.Config.r_spStabilizationTime);
           END_REGION

       END_REGION

       REGION Some faults is active

           #t_Obj_PLC.State.Error := #t_Obj_PLC.Alarm.SensorErr
           OR #t_Obj_PLC.Alarm.InverterErr
           OR #t_Obj_PLC.Alarm.PIDErr
           OR #t_Obj_PLC.Alarm.EstopHMI
           OR #t_Obj_PLC.Alarm.ExtError
           OR #t_Obj_PLC.Alarm.StabilizationErr;

           #t_Obj_PLC.Alarm.Error := #t_Obj_PLC.State.Error;
       END_REGION

   END_REGION
   //---------------------------------------------------------------
   //---------------------------------------------------------------
   REGION Release for start in any mode
       #t_ReleaseStart := NOT (#t_Obj_PLC.Alarm.SensorErr
       OR #t_Obj_PLC.Alarm.PIDErr
       OR #t_Obj_PLC.Alarm.EstopHMI
       OR #t_Obj_PLC.Alarm.ExtError)
       AND NOT #t_Obj_PLC.Mode.Disable
     //  AND NOT #t_Obj_PLC.Mode.Repair
       AND NOT #s_EdgeSim.QB_EdgeNeg
       AND NOT #t_Obj_PLC.State.FTCActive
       AND NOT #t_Obj_PLC.State.FTOActive
       AND NOT #I_Initialization;

       #s_ErrForSwitchToOff :=  NOT #t_ReleaseStart;
   END_REGION
   //---------------------------------------------------------------
   //---------------------------------------------------------------
   REGION General states
       IF NOT #t_Obj_PLC.Mode.Disable
           AND NOT #t_Obj_PLC.Mode.Repair
       THEN
           //General states 
           #t_Obj_PLC.State.SensorErr := #I_ExternalWarning;
           #t_Obj_PLC.State.InverterErr := #t_Obj_PLC.Alarm.InverterErr;
           #t_Obj_PLC.State.PIDErr := #t_Obj_PLC.Alarm.PIDErr;
           #t_Obj_PLC.State.HLActive := #t_Obj_PLC.Alarm.HLActive;
           #t_Obj_PLC.State.LLActive := #t_Obj_PLC.Alarm.LLActive;
           #t_Obj_PLC.State.DirectMode := #t_Obj_HMI.Config.b.DirectMode;
           #t_Obj_PLC.State.AllInAuto := (#t_AutoControl_Pumps.Arr[0].AutoControl_P.Mode.Auto
           OR NOT #t_AutoControl_Pumps.Arr[0].Enabled)
           AND (#t_AutoControl_Pumps.Arr[1].AutoControl_P.Mode.Auto
           OR NOT #t_AutoControl_Pumps.Arr[1].Enabled)
           AND (#t_AutoControl_Pumps.Arr[2].AutoControl_P.Mode.Auto
           OR NOT #t_AutoControl_Pumps.Arr[2].Enabled);
           #t_Obj_PLC.State.StabilizationErr := #t_Obj_PLC.Alarm.StabilizationErr;
       END_IF;

       //States for all modes
       #t_Obj_PLC.Alarm.Disable := #t_Obj_PLC.Mode.Disable;
       #t_Obj_PLC.Alarm.ManualRemote := #t_Obj_PLC.Mode.ManualRemote;
       #t_Obj_PLC.Alarm.Auto := #t_Obj_PLC.Mode.Auto;
       #t_Obj_PLC.Alarm.ManualLocal := #t_Obj_PLC.Mode.ManualLocal;
       #t_Obj_PLC.Alarm.Service := #t_Obj_PLC.Mode.Service;
       #t_Obj_PLC.Alarm.RepairOn := #t_Obj_PLC.Mode.Repair;
       #t_Obj_PLC.Alarm.IndependentOn := #t_Obj_PLC.Mode.Independent;
       #t_Obj_PLC.Alarm.SimulationOn := #t_Obj_PLC.Mode.Simulation;
       #t_Obj_PLC.Alarm.RepairOff := NOT #t_Obj_PLC.Mode.Repair;
       #t_Obj_PLC.Alarm.IndependentOff := NOT #t_Obj_PLC.Mode.Independent;
       #t_Obj_PLC.Alarm.SimulationOff := NOT #t_Obj_PLC.Mode.Simulation;

       REGION Pulses for new states
           #s_EdgeError(IB_Initialisation := #I_Initialization,
                        IB_Input := #t_Obj_PLC.State.Error);
           #s_EdgeWarning(IB_Initialisation := #I_Initialization,
                          IB_Input := false);
       END_REGION
   END_REGION
   //---------------------------------------------------------------
   //---------------------------------------------------------------
   REGION Write STW and Alarm bits into words

       //Wrapping Alarm bits in words
       #t_InternalData.di_Tmp := 0;
       #t_InternalData.i_Tmp := Serialize(SRC_VARIABLE := #t_Obj_PLC.Alarm, DEST_ARRAY => #t_Buffer, POS := #t_InternalData.di_Tmp);
       #t_Obj_HMI.Status.w_ALW1.%B0 := #t_Buffer[0];
       #t_Obj_HMI.Status.w_ALW1.%B1 := #t_Buffer[1];
       #t_Obj_HMI.Status.w_ALW2.%B0 := #t_Buffer[2];
       #t_Obj_HMI.Status.w_ALW2.%B1 := #t_Buffer[3];
       #t_Obj_HMI.Status.w_ALW3.%B0 := #t_Buffer[4];
       #t_Obj_HMI.Status.w_ALW3.%B1 := #t_Buffer[5];
       #t_Obj_HMI.Status.w_ALW4.%B0 := #t_Buffer[6];
       #t_Obj_HMI.Status.w_ALW4.%B1 := #t_Buffer[7];

       //Wrapping STW bits
       //States
       #t_InternalData.di_Tmp := 0;
       #t_InternalData.i_Tmp := Serialize(SRC_VARIABLE := #t_Obj_PLC.State, DEST_ARRAY => #t_Buffer, POS := #t_InternalData.di_Tmp);

       //Modes
       #t_InternalData.di_Tmp := 5;
       #t_InternalData.i_Tmp := Serialize(SRC_VARIABLE := #t_Obj_PLC.Mode, DEST_ARRAY => #t_Buffer, POS := #t_InternalData.di_Tmp);

       #t_Obj_HMI.Status.dw_STW.%B0 := #t_Buffer[0]; //States W1
       #t_Obj_HMI.Status.dw_STW.%B1 := #t_Buffer[1]; //States W2
       #t_Obj_HMI.Status.dw_STW.%B2 := #t_Buffer[2] OR #t_Buffer[5]; //Modes W1
       #t_Obj_HMI.Status.dw_STW.%B3 := #t_Buffer[6]; //Modes W2

   END_REGION
   //---------------------------------------------------------------
   //---------------------------------------------------------------
   REGION Write data to HMI and BUp storage
       //HMI data
       #t_Obj_HMI.i_ID := #II_Obj_ID;
       #t_Obj_HMI.i_CLSID := 151;

       //BUp retain data
       //Read retain data if initialization is active
       IF NOT #I_Initialization
       THEN
           #s_Obj_Retain_BUp.Config := #t_Obj_HMI.Config;
           #s_Obj_Retain_BUp.Counters := #t_Obj_HMI.Counters;
           #s_Obj_Retain_BUp.Mode := #t_Obj_PLC.Mode;
       END_IF;
   END_REGION
   //---------------------------------------------------------------
   //---------------------------------------------------------------
   REGION Wrap data for automode module
       #t_AutoControl.STW_HMI := #t_InternalData.d_Alw0;
       #t_AutoControl.STW := #t_InternalData.d_Alw0;

       #t_AutoControl.Mode := #t_Obj_PLC.Mode;
       #t_AutoControl.CLSID := #t_Obj_HMI.i_CLSID;
       #t_AutoControl.StatusGen.Fault := #t_Obj_PLC.State.Error;
       #t_AutoControl.StatusGen.Ready := #t_ReleaseStart;
       #t_AutoControl.StatusGen.ControlAchieve := true;

       #t_InternalData.di_Tmp := 0;
       #t_InternalData.i_Tmp := Serialize(SRC_VARIABLE := #t_AutoControl.StatusGen, DEST_ARRAY => #t_Buffer, POS := #t_InternalData.di_Tmp);
       #t_InternalData.di_Tmp := 2;
       #t_InternalData.i_Tmp := Serialize(SRC_VARIABLE := #t_AutoControl.Mode, DEST_ARRAY => #t_Buffer, POS := #t_InternalData.di_Tmp);

       #t_AutoControl.STW_HMI.%B0 := #t_Buffer[0];
       #t_AutoControl.STW_HMI.%B1 := #t_Buffer[1];
       #t_AutoControl.STW_HMI.%B2 := #t_Buffer[2];
       #t_AutoControl.STW_HMI.%B3 := #t_Buffer[3];
       #t_AutoControl.STW_HMI.%X16 := false;
   END_REGION
   //---------------------------------------------------------------
   //---------------------------------------------------------------
   REGION Write status data to HMI
       #t_Obj_HMI.Config.r_Out_MaxValue := ABS(#IR_MaxOut);
       #t_Obj_HMI.Config.r_Out_MinValue := ABS(#IR_MinOut);
       #t_Obj_HMI.Config.r_PV_MaxValue := #t_SensorObj_HMI.Config.r_MaxVal;
       #t_Obj_HMI.Config.r_PV_MinValue := #t_SensorObj_HMI.Config.r_MinVal;
       #t_Obj_HMI.Config.r_ActSpeedSP_P1 := #t_Pump1_Obj_HMI.Status.r_SetpointSpeed;
       #t_Obj_HMI.Config.r_ActSpeedSP_P2 := #t_Pump2_Obj_HMI.Status.r_SetpointSpeed;
       #t_Obj_HMI.Config.r_ActSpeedSP_P3 := #t_Pump3_Obj_HMI.Status.r_SetpointSpeed;
       #t_Obj_HMI.Config.r_ActSpeedPV_P1 := #t_Pump1_Obj_HMI.Status.r_ActualSpeed;
       #t_Obj_HMI.Config.r_ActSpeedPV_P2 := #t_Pump2_Obj_HMI.Status.r_ActualSpeed;
       #t_Obj_HMI.Config.r_ActSpeedPV_P3 := #t_Pump3_Obj_HMI.Status.r_ActualSpeed;
       #t_Obj_HMI.Config.r_Motohours_P1 := #t_Pump1_Obj_HMI.Counters.di_TimeOper_Tot;
       #t_Obj_HMI.Config.r_Motohours_P2 := #t_Pump2_Obj_HMI.Counters.di_TimeOper_Tot;
       #t_Obj_HMI.Config.r_Motohours_P3 := #t_Pump3_Obj_HMI.Counters.di_TimeOper_Tot;
       #t_Obj_HMI.Config.r_PV_ActValue := #t_Obj_PIDCon.r_Input;
       #t_Obj_HMI.Config.r_Out_ActValue := ABS(#t_Obj_PIDCon.r_Output);

       #t_Obj_HMI.Status.dw_STW_PID := #t_Obj_PIDCon.dw_ErrorBits;

       #t_Obj_HMI.Status.dw_STW_P1.%X0 := #t_Pump1_Obj_HMI.Status.dw_STW.%X4;
       #t_Obj_HMI.Status.dw_STW_P1.%X1 := #t_Pump1_Obj_HMI.Status.dw_STW.%X6;
       #t_Obj_HMI.Status.dw_STW_P1.%X2 := #t_Obj_HMI.Config.b.Enabled_P1;
       #t_Obj_HMI.Status.dw_STW_P1.%X3 := #t_Pump1_Obj_HMI.Status.dw_STW.%X25;

       #t_Obj_HMI.Status.dw_STW_P2.%X0 := #t_Pump2_Obj_HMI.Status.dw_STW.%X4;
       #t_Obj_HMI.Status.dw_STW_P2.%X1 := #t_Pump2_Obj_HMI.Status.dw_STW.%X6;
       #t_Obj_HMI.Status.dw_STW_P2.%X2 := #t_Obj_HMI.Config.b.Enabled_P2;
       #t_Obj_HMI.Status.dw_STW_P2.%X3 := #t_Pump2_Obj_HMI.Status.dw_STW.%X25;

       #t_Obj_HMI.Status.dw_STW_P3.%X0 := #t_Pump3_Obj_HMI.Status.dw_STW.%X4;
       #t_Obj_HMI.Status.dw_STW_P3.%X1 := #t_Pump3_Obj_HMI.Status.dw_STW.%X6;
       #t_Obj_HMI.Status.dw_STW_P3.%X2 := #t_Obj_HMI.Config.b.Enabled_P3;
       #t_Obj_HMI.Status.dw_STW_P3.%X3 := #t_Pump3_Obj_HMI.Status.dw_STW.%X25;

   END_REGION
   //---------------------------------------------------------------
   //---------------------------------------------------------------
   REGION Write data to out DB
       //Write data  PLC
       VariantPut(SRC := #t_PLC_CycleInfo,
                  DST := #IQ_PLC_CycleInfo);

       //Write Object data
       //DB num 
       IF #II_Obj_ID >= 0
           AND NOT #t_DataErr
       THEN
           //Write HMI data
           VariantPut(SRC := #t_Obj_HMI,
                      DST := #t_ObjVar_HMI);

           //Write PLC data
           VariantPut(SRC := #t_Obj_PLC,
                      DST := #t_ObjVar_PLC);

           //Write PID data
           VariantPut(SRC := #t_Obj_PIDCon,
                      DST := #t_ObjVar_PIDCon);
       ELSE
           #t_DataErr := true;
       END_IF;

       //Write pumps data
       IF #IA_ID_Inv[0] >= 0
           AND NOT #t_DataErr
       THEN
           REGION Pump 1
               "DB_AutoControl_arr".AutoControl_arr[#IA_ID_Inv[0]] := #t_AutoControl_Pumps.Arr[0].AutoControl_P;
           END_REGION

       ELSE
           #t_DataErr := true;
       END_IF;

       IF #IA_ID_Inv[1] >= 0
           AND NOT #t_DataErr
       THEN
           REGION Pump 2
               "DB_AutoControl_arr".AutoControl_arr[#IA_ID_Inv[1]] := #t_AutoControl_Pumps.Arr[1].AutoControl_P;
           END_REGION

       ELSE
           #t_DataErr := true;
       END_IF;

       IF #IA_ID_Inv[2] >= 0
           AND NOT #t_DataErr
       THEN
           REGION Pump 3
               "DB_AutoControl_arr".AutoControl_arr[#IA_ID_Inv[2]] := #t_AutoControl_Pumps.Arr[2].AutoControl_P;
           END_REGION
       ELSE
           #t_DataErr := true;
       END_IF;

       //Write general info data
       CASE #II_Obj_ID OF
           0..999:  // ID of element in range
               "DB_AutoControl_arr".AutoControl_arr[#II_Obj_ID] := #t_AutoControl;
           ELSE
               ;
       END_CASE;

   END_REGION
   //---------------------------------------------------------------
   //---------------------------------------------------------------
   REGION Outputs of block
       #QR_Out_PID := #t_Obj_PIDCon.r_Output;
       #QI_Out_PID := #t_Obj_PIDCon.OutPER;
       #Q_CmdPWM := #t_Obj_PIDCon.OutPWM;
       #Q_Reset := #t_ResetLogic;
       #Q_Error := #t_Obj_PLC.State.Error;
       #Q_Auto := #t_Obj_PLC.Mode.Auto;
       #Q_DataErr := #t_DataErr;
   END_REGION

   //Test text 17.02.2022
   //Old Code 06.28.2022
   (*
   REGION Define current, next and prev points
           //Some of pumps is running
           #t_SomePumpIsRunning := #t_Pump1_Obj_HMI.Status.dw_STW.%X6
           OR #t_Pump2_Obj_HMI.Status.dw_STW.%X6
           OR #t_Pump3_Obj_HMI.Status.dw_STW.%X6;

           IF NOT #t_SomePumpIsRunning
           THEN
               #si_CurrentPoint := -1;
               FOR #ti_Cnt := 0 TO 2 DO
                   IF #t_AutoControl_Pumps.Arr[#ti_Cnt].i_Priority = 1
                       AND #t_AutoControl_Pumps.Arr[#ti_Cnt].Enabled
                   THEN
                       #si_CurrentPoint := #t_AutoControl_Pumps.Arr[#ti_Cnt].i_Priority;
                   END_IF;
               END_FOR;
           ELSE
               //Define points for go up
               IF #s_EdgeUp.QB_EdgePos
               THEN
                   #si_CurrentPoint := #si_CurrentPoint;
                   FOR #ti_Cnt := 0 TO 2 DO
                       IF #t_AutoControl_Pumps.Arr[#ti_Cnt].i_Priority >= (#si_CurrentPoint + 1)
                           AND #t_AutoControl_Pumps.Arr[#ti_Cnt].Enabled
                           AND #t_AutoControl_Pumps.Arr[#ti_Cnt].AutoControl_P.STW_HMI.%X25
                           AND #t_AutoControl_Pumps.Arr[#ti_Cnt].AutoControl_P.STW_HMI.%X1
                       THEN
                           #si_CurrentPoint := #t_AutoControl_Pumps.Arr[#ti_Cnt].i_Priority;
                           #t_Obj_PIDCon.r_IntegralSum := #IR_MinOut - #t_Obj_PIDCon.r_Gain * (#t_Obj_PIDCon.r_Setpoint - #t_Obj_PIDCon.r_Input);
                           #tr_PID_Out := #IR_MinOut;
                           #t_Obj_PIDCon.SetIntegralSum := true;
                           EXIT;
                       END_IF;
                   END_FOR;
               END_IF;

               //Define points for go dwn
               IF #s_EdgeDwn.QB_EdgePos
               THEN
                   #si_CurrentPoint := #si_CurrentPoint;
                   FOR #ti_Cnt := 0 TO 2 DO
                       IF #t_AutoControl_Pumps.Arr[#ti_Cnt].i_Priority <= (#si_CurrentPoint - 1)
                           AND #t_AutoControl_Pumps.Arr[#ti_Cnt].Enabled
                           AND #t_AutoControl_Pumps.Arr[#ti_Cnt].AutoControl_P.STW_HMI.%X25
                           AND #t_AutoControl_Pumps.Arr[#ti_Cnt].AutoControl_P.STW_HMI.%X1
                       THEN
                           #si_CurrentPoint := #t_AutoControl_Pumps.Arr[#ti_Cnt].i_Priority;
                           #t_Obj_PIDCon.r_IntegralSum := #IR_MaxOut - #t_Obj_PIDCon.r_Gain * (#t_Obj_PIDCon.r_Setpoint - #t_Obj_PIDCon.r_Input);
                           #tr_PID_Out := #IR_MaxOut;
                           #t_Obj_PIDCon.SetIntegralSum := true;
                           EXIT;
                       END_IF;
                   END_FOR;
               END_IF;
           END_IF;
       END_REGION
   *)
END_FUNCTION_BLOCK
